TYPE DS_fbStationSequenceRecipeStore : (*Full Occupied Byte = 500*)
STRUCT

	bCopyPB : BOOL; (* Byte "n" *)
	sReservedBool : STRING(50); (* Byte "n+1~n+99" *)


	iStationSequenceRecipeNo: INT; (* Byte "n+100, n+101" *)	(* 10 sets of Station Sequence Recipe *)
	iCopyToSubRecipeNo : INT; (* Byte "n+102, n+103" *)
	sReservedInt : STRING(50); (* Byte "n+104~n+199" *)


	sStationSequenceRecipeDescription : STRING(50); (* Byte "n+200~n+299" *)  (* Description of Station Sequence Recipe - Naming*)


	DsStationSequenceRecipeMemory : DS_StationSequenceRecipeMemory; (* Byte "n+300 onward" *)






END_STRUCT
END_TYPE

(* stored: Version 1.1.0.1, ProductVersion 3.1.4024.12
   DUT DS_fbStationSequenceRecipeStore: Id {ce70b5c0-d815-49e4-a0f4-7f32089f3776} *)
